INTERFACE IDifferentiable EXTENDS IOut

METHOD Control: IOut
VAR_INPUT
    setpoint : LREAL;
END_VAR
END_METHOD

METHOD Iir : IBaseSignal
VAR_INPUT
    decay : LREAL;
END_VAR
END_METHOD

METHOD Update : ISignal
VAR_INPUT
    value : LREAL;
END_VAR
END_METHOD

END_INTERFACE

(* stored: Version 1.1.0.1, ProductVersion 3.1.4024.12
   Itf IDifferentiable: Id {ef3bce93-b4be-41da-891f-48a7afa41e3d}
   Method Control: Id {629d8683-07d5-4dca-9fe9-930d2298bc20}
   Method Iir: Id {8fd6cd0c-7c2a-4af0-8c7a-f34c2613fe30}
   Method Update: Id {a5b00a30-c45e-4d64-88f3-9feef6670dfc} *)
